TYPE ST_DataLog :
STRUCT
  WorkOrder : WORD;
  Duration  : REAL; // [ms]
  Position  : REAL;
END_STRUCT
END_TYPE

(* stored: Version 1.1.0.1, ProductVersion 3.1.4022.18
   DUT ST_DataLog: Id {f4754bca-372b-410d-b85c-0a13b5d980eb} *)
